// TIA Portal V19 export
VAR_GLOBAL   // PLC tag table "LB308"
   LB308_Scarico_Interno_SX_Pb_Aux2 AT %I351.4 : Bool;   // 351SH2
   LB308_Scarico_Interno_SX_Pb_Aux1 AT %I351.3 : Bool;   // 351SH1
   LB308_Scarico_Interno_SX_Lp_Aux2 AT %Q351.4 : Bool;   // 351SH2
   LB308_Scarico_Interno_SX_Lp_Aux1 AT %Q351.3 : Bool;   // 351SH1
END_VAR
